KUKA KRL program: Rack_Azul_Cerrar_PLC.src, Rack_Azul_Cerrar_PLC.dat

--- Rack_Azul_Cerrar_PLC.src ---
&ACCESS RVO1
&REL 14
&COMMENT CERRAR BANDEJAS PLC
&PARAM EDITMASK = *
&PARAM TEMPLATE = C:\KRC\Roboter\Template\vorgabe
&PARAM DISKPATH = KRC:\R1\Program\MAFELEC
DEF Rack_Azul_Cerrar_PLC( )
;FOLD INI;%{PE}
  ;FOLD BASISTECH INI
    GLOBAL INTERRUPT DECL 3 WHEN $STOPMESS==TRUE DO IR_STOPM ( )
    INTERRUPT ON 3
    BAS (#INITMOV,0 )
  ;ENDFOLD (BASISTECH INI)
;FOLD SPOTTECH INI
USERSPOT(#INIT)
;ENDFOLD (SPOTTECH INI)
;FOLD GRIPPERTECH INI
USER_GRP(0,DUMMY,DUMMY,GDEFAULT)
;ENDFOLD (GRIPPERTECH INI)
  ;FOLD USER INI
    ;Make your modifications here
INTERRUPT DECL 82 WHEN I_121R1S501 DO STOP_PUSH ()
INTERRUPT DECL 92 WHEN I_121R1S501 DO STOP_PUSH ()

  ;ENDFOLD (USER INI)
;ENDFOLD (INI)
;################################################
; PROYECTO: MAFELEC PLANTA DE BATERIAS
; ROBOT: 121_R1
; PROGRAMA: CERRAR BANDEJAS EN RACK AZUL
; CREADO POR: Alejandro Company(zaisor robotics)
; FECHA: 23-NOVIEMBRE-2022
; MODIFICADO POR:
; FECHA MODIFICACION: 05-ENERO-2023
;################################################

;FOLD PTP HOME Vel=100 % PDAT1;%{PE}%R 8.3.48,%MKUKATPBASIS,%CMOVE,%VPTP,%P 1:PTP, 2:HOME, 3:, 5:100, 7:PDAT1
$BWDSTART=FALSE
PDAT_ACT=PPDAT1
FDAT_ACT=FHOME
BAS(#PTP_PARAMS,100)
$H_POS=XHOME
PTP XHOME
;ENDFOLD
; POSICION DE ESPERA ENTRADA RACK 2 (AZUL)
;FOLD PTP POS_ESPERA_AREA2 Vel=50 % H Tool[9]:T_Gripper1_Vacio Base[0];%{PE}%R 8.3.48,%MKUKATPBASIS,%CMOVE,%VPTP,%P 1:PTP, 2:POS_ESPERA_AREA2, 3:, 5:50, 7:H
$BWDSTART=FALSE
PDAT_ACT=PH
FDAT_ACT=FPOS_ESPERA_AREA2
BAS(#PTP_PARAMS,50)
PTP XPOS_ESPERA_AREA2
;ENDFOLD
;ESPERA AREA 2
WAIT FOR I_ARDY_2
O_AREL_2=FALSE

WAIT FOR I_121R1S1000==FALSE

;FOLD PTP P_CERRAR10 CONT Vel=50 % H Tool[2]:T_PUSH2 Base[2]:Rack_Azul;%{PE}%R 8.3.48,%MKUKATPBASIS,%CMOVE,%VPTP,%P 1:PTP, 2:P_CERRAR10, 3:C_DIS, 5:50, 7:H
$BWDSTART=FALSE
PDAT_ACT=PH
FDAT_ACT=FP_CERRAR10
BAS(#PTP_PARAMS,50)
PTP XP_CERRAR10 C_DIS
;ENDFOLD

INI_BUCLE:
;FOLD PTP P10 Vel=50 % H Tool[2]:T_PUSH2 Base[2]:Rack_Azul;%{PE}%R 8.3.48,%MKUKATPBASIS,%CMOVE,%VPTP,%P 1:PTP, 2:P10, 3:, 5:50, 7:H
$BWDSTART=FALSE
PDAT_ACT=PH
FDAT_ACT=FP10
BAS(#PTP_PARAMS,50)
PTP XP10
;ENDFOLD

RA_Bandeja_Nr=0
O_TYPE_RQ=TRUE
WAIT FOR (I_TYPE_INFO > 20) AND (I_TYPE_INFO < 26)
RA_Bandeja_Nr=I_TYPE_INFO

Rack_Azul_Cerrar_D ()

END
DEF STOP_PUSH()
INTERRUPT OFF 82
INTERRUPT OFF 92

BRAKE
WAIT SEC 0
PTP $POS_ACT
LIN $POS_INT
$OV_PRO=OLD_OVPRO

;RESUME

END

--- Rack_Azul_Cerrar_PLC.dat ---
&ACCESS RVO1
&REL 14
&COMMENT CERRAR BANDEJAS PLC
&PARAM EDITMASK = *
&PARAM TEMPLATE = C:\KRC\Roboter\Template\vorgabe
&PARAM DISKPATH = KRC:\R1\Program\MAFELEC
DEFDAT  Rack_Azul_Cerrar_PLC
;FOLD EXTERNAL DECLARATIONS;%{PE}%MKUKATPBASIS,%CEXT,%VCOMMON,%P
;FOLD GRIPPERTECH EXT
EXT  H50 (INT  :IN,INT  :IN,INT  :IN,GRP_TYP  :IN )
;ENDFOLD (GRIPPERTECH EXT)
;FOLD SPOTTECH EXT
EXT  USERSPOT (S_COMMAND  :IN,SPOT_TYPE  :IN )
;ENDFOLD (SPOTTECH EXT)
;FOLD BASISTECH EXT;%{PE}%MKUKATPBASIS,%CEXT,%VEXT,%P
EXT  BAS (BAS_COMMAND  :IN,REAL  :IN )
DECL INT SUCCESS
;ENDFOLD (BASISTECH EXT)
;FOLD USER EXT;%{E}%MKUKATPUSER,%CEXT,%VEXT,%P
;Make your modifications here

;ENDFOLD (USER EXT)
;ENDFOLD (EXTERNAL DECLARATIONS)
DECL BASIS_SUGG_T LAST_BASIS={POINT1[] "HOME                    ",POINT2[] "HOME                    ",CP_PARAMS[] "CPDAT0                  ",PTP_PARAMS[] "PDAT1                   ",CONT[] "                        ",CP_VEL[] "2.0                     ",PTP_VEL[] "100                     ",SYNC_PARAMS[] "SYNCDAT                 ",SPL_NAME[] "S0                      ",A_PARAMS[] "ADAT0                   "}
DECL PDAT PH={VEL 100.000,ACC 100.000,APO_DIST 100.000,APO_MODE #CDIS,GEAR_JERK 50.0000,EXAX_IGN 0}
DECL E6POS XPOS_ESPERA_AREA1={X 112.943756,Y -227.851166,Z 2716.11304,A 36.2463837,B -15.5853510,C 56.0520973,S 3,T 42,E1 0.0,E2 0.0,E3 0.0,E4 0.0,E5 0.0,E6 0.0}
DECL FDAT FPOS_ESPERA_AREA1={TOOL_NO 9,BASE_NO 0,IPO_FRAME #BASE,POINT2[] " ",TQ_STATE FALSE}
DECL LDAT LL={VEL 2.00000,ACC 25.0000,APO_DIST 25.0000,APO_FAC 50.0000,AXIS_VEL 100.000,AXIS_ACC 100.000,ORI_TYP #VAR,CIRC_TYP #BASE,JERK_FAC 50.0000,GEAR_JERK 50.0000,EXAX_IGN 0}
DECL E6POS XPOS_AREA1_LIBRE={X -250.533554,Y -43.6507149,Z 2716.11304,A -84.6604385,B 6.50295877,C 57.2217522,S 3,T 42,E1 0.0,E2 0.0,E3 0.0,E4 0.0,E5 0.0,E6 0.0}
DECL FDAT FPOS_AREA1_LIBRE={TOOL_NO 9,BASE_NO 0,IPO_FRAME #BASE,POINT2[] " ",TQ_STATE FALSE}
DECL E6POS XP111={X 557.799622,Y -753.947571,Z -222.785736,A -88.9974060,B 13.7721291,C 89.1738281,S 6,T 58,E1 0.0,E2 0.0,E3 0.0,E4 0.0,E5 0.0,E6 0.0}
DECL FDAT FP111={TOOL_NO 1,BASE_NO 1,IPO_FRAME #BASE,POINT2[] " ",TQ_STATE FALSE}
DECL E6POS XP10={X 1430.18262,Y 33.1879578,Z 909.224609,A 86.6829224,B -17.0911541,C -157.124573,S 2,T 35,E1 0.0,E2 0.0,E3 0.0,E4 0.0,E5 0.0,E6 0.0}
DECL FDAT FP10={TOOL_NO 2,BASE_NO 2,IPO_FRAME #BASE,POINT2[] " ",TQ_STATE FALSE}
DECL E6POS XP110={X 632.645691,Y 303.475861,Z -186.174820,A -88.8950272,B 31.1322117,C 89.5053635,S 6,T 58,E1 0.0,E2 0.0,E3 0.0,E4 0.0,E5 0.0,E6 0.0}
DECL FDAT FP110={TOOL_NO 1,BASE_NO 1,IPO_FRAME #BASE,POINT2[] " ",TQ_STATE FALSE}
DECL E6POS XP120={X 535.775818,Y 225.276917,Z -536.621948,A -91.0083771,B 14.9493265,C 94.2730637,S 6,T 58,E1 0.0,E2 0.0,E3 0.0,E4 0.0,E5 0.0,E6 0.0}
DECL FDAT FP120={TOOL_NO 1,BASE_NO 1,IPO_FRAME #BASE,POINT2[] " ",TQ_STATE FALSE}
DECL E6POS XP_ABRIR10={X -250.533554,Y -43.6507149,Z 2716.11304,A -84.6604385,B 6.50295877,C 57.2217522,S 3,T 42,E1 0.0,E2 0.0,E3 0.0,E4 0.0,E5 0.0,E6 0.0}
DECL FDAT FP_ABRIR10={TOOL_NO 9,BASE_NO 0,IPO_FRAME #BASE,POINT2[] " ",TQ_STATE FALSE}
DECL E6POS XP_AHOME={X 112.943756,Y -227.851166,Z 2716.11304,A 36.2463837,B -15.5853510,C 56.0520973,S 3,T 42,E1 0.0,E2 0.0,E3 0.0,E4 0.0,E5 0.0,E6 0.0}
DECL FDAT FP_aHOME={TOOL_NO 9,BASE_NO 0,IPO_FRAME #BASE,POINT2[] " ",TQ_STATE FALSE}
DECL E6POS XIni_Cerrar_B1={X 557.764587,Y -781.945251,Z -181.205933,A -89.0119858,B 10.6981707,C 89.1186752,S 6,T 58,E1 0.0,E2 0.0,E3 0.0,E4 0.0,E5 0.0,E6 0.0}
DECL FDAT FIni_Cerrar_B1={TOOL_NO 1,BASE_NO 1,IPO_FRAME #BASE,POINT2[] " ",TQ_STATE FALSE}
DECL E6POS XAux_Cerrar_B1={X 557.840454,Y -622.833801,Z -384.869720,A -88.9527512,B 18.9294662,C 89.2742310,S 6,T 58,E1 0.0,E2 0.0,E3 0.0,E4 0.0,E5 0.0,E6 0.0}
DECL E6POS XFin_Cerrar_B1={X 558.459229,Y -381.955719,Z -941.239441,A -88.7644653,B 34.8009872,C 89.6337738,S 6,T 58,E1 0.0,E2 0.0,E3 0.0,E4 0.0,E5 0.0,E6 0.0}
DECL FDAT FFin_Cerrar_B1={TOOL_NO 1,BASE_NO 1,IPO_FRAME #BASE,POINT2[] "XAux_Cerrar_B1",TQ_STATE FALSE}
DECL E6POS XP0={X 632.645691,Y 303.475861,Z -186.174820,A -88.8950272,B 31.1322117,C 89.5053635,S 6,T 58,E1 0.0,E2 0.0,E3 0.0,E4 0.0,E5 0.0,E6 0.0}
DECL FDAT FP0={TOOL_NO 1,BASE_NO 1,IPO_FRAME #BASE,POINT2[] " ",TQ_STATE FALSE}
DECL E6POS XIni_Cerrar_B2={X 633.606323,Y -740.251,Z 3.60236120,A -89.0051498,B 9.17837143,C 89.0890656,S 6,T 58,E1 0.0,E2 0.0,E3 0.0,E4 0.0,E5 0.0,E6 0.0}
DECL FDAT FIni_Cerrar_B2={TOOL_NO 1,BASE_NO 1,IPO_FRAME #BASE,POINT2[] " ",TQ_STATE FALSE}
DECL E6POS XP1={X 633.606323,Y -740.251,Z -11.7250,A -89.0051498,B 9.17837143,C 89.0890656,S 6,T 58,E1 0.0,E2 0.0,E3 0.0,E4 0.0,E5 0.0,E6 0.0}
DECL FDAT FP1={TOOL_NO 1,BASE_NO 1,IPO_FRAME #BASE,POINT2[] " ",TQ_STATE FALSE}
DECL E6POS XAux_Cerrar_B2={X 634.042603,Y -508.122833,Z -357.182983,A -88.8871536,B 26.3570118,C 89.4227295,S 6,T 58,E1 0.0,E2 0.0,E3 0.0,E4 0.0,E5 0.0,E6 0.0}
DECL E6POS XFin_Cerrar_B2={X 634.405884,Y -397.733490,Z -741.710266,A -88.8505630,B 28.6699753,C 89.4738922,S 6,T 58,E1 0.0,E2 0.0,E3 0.0,E4 0.0,E5 0.0,E6 0.0}
DECL FDAT FFin_Cerrar_B2={TOOL_NO 1,BASE_NO 1,IPO_FRAME #BASE,POINT2[] "XAux_Cerrar_B2",TQ_STATE FALSE}
DECL E6POS XP2={X 535.775818,Y 225.276917,Z -536.621948,A -91.0083771,B 14.9493265,C 94.2730637,S 6,T 58,E1 0.0,E2 0.0,E3 0.0,E4 0.0,E5 0.0,E6 0.0}
DECL FDAT FP2={TOOL_NO 1,BASE_NO 1,IPO_FRAME #BASE,POINT2[] " ",TQ_STATE FALSE}
DECL E6POS XP210={X 536.241516,Y 225.176605,Z 24.6719704,A -90.9851761,B 14.9447651,C 94.2668762,S 6,T 58,E1 0.0,E2 0.0,E3 0.0,E4 0.0,E5 0.0,E6 0.0}
DECL FDAT FP210={TOOL_NO 1,BASE_NO 1,IPO_FRAME #BASE,POINT2[] " ",TQ_STATE FALSE}
DECL E6POS XP220={X 535.775818,Y 225.276917,Z -194.099075,A -91.0083771,B 14.9493265,C 94.2730637,S 6,T 58,E1 0.0,E2 0.0,E3 0.0,E4 0.0,E5 0.0,E6 0.0}
DECL FDAT FP220={TOOL_NO 1,BASE_NO 1,IPO_FRAME #BASE,POINT2[] " ",TQ_STATE FALSE}
DECL E6POS XP3={X 536.241516,Y 225.176605,Z 24.6719704,A -90.9851761,B 14.9447651,C 94.2668762,S 6,T 58,E1 0.0,E2 0.0,E3 0.0,E4 0.0,E5 0.0,E6 0.0}
DECL FDAT FP3={TOOL_NO 1,BASE_NO 1,IPO_FRAME #BASE,POINT2[] " ",TQ_STATE FALSE}
DECL E6POS XIni_Cerrar_B3={X 587.397888,Y -796.521118,Z 250.544754,A -89.9228,B 6.59320593,C 91.5957413,S 6,T 58,E1 0.0,E2 0.0,E3 0.0,E4 0.0,E5 0.0,E6 0.0}
DECL FDAT FIni_Cerrar_B3={TOOL_NO 1,BASE_NO 1,IPO_FRAME #BASE,POINT2[] " ",TQ_STATE FALSE}
DECL E6POS XP4={X 633.606323,Y -740.251,Z -11.7250,A -89.0051498,B 9.17837143,C 89.0890656,S 6,T 58,E1 0.0,E2 0.0,E3 0.0,E4 0.0,E5 0.0,E6 0.0}
DECL FDAT FP4={TOOL_NO 1,BASE_NO 1,IPO_FRAME #BASE,POINT2[] " ",TQ_STATE FALSE}
DECL E6POS XAux_Cerrar_B3={X 587.803650,Y -538.859497,Z -87.8424835,A -89.9063950,B 15.5115423,C 91.6123123,S 6,T 58,E1 0.0,E2 0.0,E3 0.0,E4 0.0,E5 0.0,E6 0.0}
DECL E6POS XFin_Cerrar_B3={X 588.007202,Y -397.554932,Z -533.267273,A -89.8953171,B 21.9562569,C 91.6268768,S 6,T 58,E1 0.0,E2 0.0,E3 0.0,E4 0.0,E5 0.0,E6 0.0}
DECL FDAT FFin_Cerrar_B3={TOOL_NO 1,BASE_NO 1,IPO_FRAME #BASE,POINT2[] "XAux_Cerrar_B3",TQ_STATE FALSE}
DECL E6POS XP5={X 535.775818,Y 225.276917,Z -194.099075,A -91.0083771,B 14.9493265,C 94.2730637,S 6,T 58,E1 0.0,E2 0.0,E3 0.0,E4 0.0,E5 0.0,E6 0.0}
DECL FDAT FP5={TOOL_NO 1,BASE_NO 1,IPO_FRAME #BASE,POINT2[] " ",TQ_STATE FALSE}
DECL E6POS XP310={X 536.344910,Y 225.151108,Z 251.906281,A -90.9788437,B 14.9441595,C 94.2655792,S 6,T 26,E1 0.0,E2 0.0,E3 0.0,E4 0.0,E5 0.0,E6 0.0}
DECL FDAT FP310={TOOL_NO 1,BASE_NO 1,IPO_FRAME #BASE,POINT2[] " ",TQ_STATE FALSE}
DECL E6POS XP320={X 535.775818,Y 225.276917,Z -194.099075,A -91.0083771,B 14.9493265,C 94.2730637,S 6,T 58,E1 0.0,E2 0.0,E3 0.0,E4 0.0,E5 0.0,E6 0.0}
DECL FDAT FP320={TOOL_NO 1,BASE_NO 1,IPO_FRAME #BASE,POINT2[] " ",TQ_STATE FALSE}
DECL E6POS XP310_1={X 587.398743,Y -796.520813,Z 219.048569,A -89.9227676,B 6.59320068,C 91.5957413,S 6,T 58,E1 0.0,E2 0.0,E3 0.0,E4 0.0,E5 0.0,E6 0.0}
DECL FDAT FP310_1={TOOL_NO 1,BASE_NO 1,IPO_FRAME #BASE,POINT2[] " ",TQ_STATE FALSE}
DECL E6POS XP6={X 536.241516,Y 225.176605,Z 24.6719704,A -90.9851761,B 14.9447651,C 94.2668762,S 6,T 58,E1 0.0,E2 0.0,E3 0.0,E4 0.0,E5 0.0,E6 0.0}
DECL FDAT FP6={TOOL_NO 1,BASE_NO 1,IPO_FRAME #BASE,POINT2[] " ",TQ_STATE FALSE}
DECL E6POS XIni_Cerrar_B4={X 547.014465,Y -762.279480,Z 527.953308,A -92.0144501,B 13.7285652,C 90.3226547,S 6,T 26,E1 0.0,E2 0.0,E3 0.0,E4 0.0,E5 0.0,E6 0.0}
DECL FDAT FIni_Cerrar_B4={TOOL_NO 1,BASE_NO 1,IPO_FRAME #BASE,POINT2[] " ",TQ_STATE FALSE}
DECL E6POS XP7={X 633.606323,Y -740.251,Z -11.7250,A -89.0051498,B 9.17837143,C 89.0890656,S 6,T 58,E1 0.0,E2 0.0,E3 0.0,E4 0.0,E5 0.0,E6 0.0}
DECL FDAT FP7={TOOL_NO 1,BASE_NO 1,IPO_FRAME #BASE,POINT2[] " ",TQ_STATE FALSE}
DECL E6POS XAux_Cerrar_B4={X 547.619568,Y -529.437683,Z 86.4444046,A -92.0362,B 21.7243443,C 90.2498322,S 6,T 26,E1 0.0,E2 0.0,E3 0.0,E4 0.0,E5 0.0,E6 0.0}
DECL E6POS XFin_Cerrar_B4={X 547.891113,Y -426.606598,Z -334.407837,A -92.0266571,B 21.7223244,C 90.2480469,S 6,T 58,E1 0.0,E2 0.0,E3 0.0,E4 0.0,E5 0.0,E6 0.0}
DECL FDAT FFin_Cerrar_B4={TOOL_NO 1,BASE_NO 1,IPO_FRAME #BASE,POINT2[] "XAux_Cerrar_B4",TQ_STATE FALSE}
DECL E6POS XP8={X 535.775818,Y 225.276917,Z -194.099075,A -91.0083771,B 14.9493265,C 94.2730637,S 6,T 58,E1 0.0,E2 0.0,E3 0.0,E4 0.0,E5 0.0,E6 0.0}
DECL FDAT FP8={TOOL_NO 1,BASE_NO 1,IPO_FRAME #BASE,POINT2[] " ",TQ_STATE FALSE}
DECL E6POS XP410={X 546.439087,Y 225.985733,Z 608.963928,A -94.2845764,B 13.2172089,C 80.7249,S 6,T 26,E1 0.0,E2 0.0,E3 0.0,E4 0.0,E5 0.0,E6 0.0}
DECL FDAT FP410={TOOL_NO 1,BASE_NO 1,IPO_FRAME #BASE,POINT2[] " ",TQ_STATE FALSE}
DECL E6POS XP410_1={X 547.319458,Y -761.898315,Z 410.812561,A -92.0465546,B 21.7247772,C 90.2501144,S 6,T 26,E1 0.0,E2 0.0,E3 0.0,E4 0.0,E5 0.0,E6 0.0}
DECL FDAT FP410_1={TOOL_NO 1,BASE_NO 1,IPO_FRAME #BASE,POINT2[] " ",TQ_STATE FALSE}
DECL E6POS XP420={X 525.192,Y 187.708069,Z 115.738434,A -91.6678391,B 6.13838816,C 94.1520309,S 6,T 58,E1 0.0,E2 0.0,E3 0.0,E4 0.0,E5 0.0,E6 0.0}
DECL FDAT FP420={TOOL_NO 1,BASE_NO 1,IPO_FRAME #BASE,POINT2[] " ",TQ_STATE FALSE}
DECL E6POS XP9={X 536.241516,Y 225.176605,Z 24.6719704,A -90.9851761,B 14.9447651,C 94.2668762,S 6,T 58,E1 0.0,E2 0.0,E3 0.0,E4 0.0,E5 0.0,E6 0.0}
DECL FDAT FP9={TOOL_NO 1,BASE_NO 1,IPO_FRAME #BASE,POINT2[] " ",TQ_STATE FALSE}
DECL E6POS XIni_Cerrar_B5={X 644.333130,Y -771.042114,Z 1009.38544,A -93.7095184,B 18.5084820,C 84.4919510,S 6,T 26,E1 0.0,E2 0.0,E3 0.0,E4 0.0,E5 0.0,E6 0.0}
DECL FDAT FIni_Cerrar_B5={TOOL_NO 1,BASE_NO 1,IPO_FRAME #BASE,POINT2[] " ",TQ_STATE FALSE}
DECL E6POS XP11={X 633.606323,Y -740.251,Z -11.7250,A -89.0051498,B 9.17837143,C 89.0890656,S 6,T 58,E1 0.0,E2 0.0,E3 0.0,E4 0.0,E5 0.0,E6 0.0}
DECL FDAT FP11={TOOL_NO 1,BASE_NO 1,IPO_FRAME #BASE,POINT2[] " ",TQ_STATE FALSE}
DECL E6POS XAux_Cerrar_B5={X 645.412,Y -297.960297,Z 334.856628,A -91.5430527,B 23.7528038,C 84.3394470,S 6,T 26,E1 0.0,E2 0.0,E3 0.0,E4 0.0,E5 0.0,E6 0.0}
DECL E6POS XFin_Cerrar_B5={X 647.239136,Y -199.588867,Z -115.631508,A -87.2260361,B 11.0592718,C 90.0945892,S 6,T 58,E1 0.0,E2 0.0,E3 0.0,E4 0.0,E5 0.0,E6 0.0}
DECL FDAT FFin_Cerrar_B5={TOOL_NO 1,BASE_NO 1,IPO_FRAME #BASE,POINT2[] "XAux_Cerrar_B5",TQ_STATE FALSE}
DECL E6POS XP12={X 535.775818,Y 225.276917,Z -194.099075,A -91.0083771,B 14.9493265,C 94.2730637,S 6,T 58,E1 0.0,E2 0.0,E3 0.0,E4 0.0,E5 0.0,E6 0.0}
DECL FDAT FP12={TOOL_NO 1,BASE_NO 1,IPO_FRAME #BASE,POINT2[] " ",TQ_STATE FALSE}
DECL E6POS XP510={X 642.977051,Y 234.134598,Z 1082.35,A -97.9549866,B 9.71833515,C 62.4231300,S 6,T 26,E1 0.0,E2 0.0,E3 0.0,E4 0.0,E5 0.0,E6 0.0}
DECL FDAT FP510={TOOL_NO 1,BASE_NO 1,IPO_FRAME #BASE,POINT2[] " ",TQ_STATE FALSE}
DECL E6POS XP510_1={X 644.512329,Y -684.707275,Z 831.107483,A -91.5230255,B 18.5093899,C 84.4910736,S 6,T 26,E1 0.0,E2 0.0,E3 0.0,E4 0.0,E5 0.0,E6 0.0}
DECL FDAT FP510_1={TOOL_NO 1,BASE_NO 1,IPO_FRAME #BASE,POINT2[] " ",TQ_STATE FALSE}
DECL E6POS XP520={X 536.730957,Y 225.074142,Z 89.3547668,A -90.9613,B 14.9400396,C 94.2604446,S 6,T 58,E1 0.0,E2 0.0,E3 0.0,E4 0.0,E5 0.0,E6 0.0}
DECL FDAT FP520={TOOL_NO 1,BASE_NO 1,IPO_FRAME #BASE,POINT2[] " ",TQ_STATE FALSE}
DECL E6POS XP210_1={X 633.606323,Y -740.251,Z -11.7250,A -89.0051498,B 9.17837143,C 89.0890656,S 6,T 58,E1 0.0,E2 0.0,E3 0.0,E4 0.0,E5 0.0,E6 0.0}
DECL FDAT FP210_1={TOOL_NO 1,BASE_NO 1,IPO_FRAME #BASE,POINT2[] " ",TQ_STATE FALSE}
DECL E6POS XP110_1={X 557.799622,Y -753.947571,Z -222.785736,A -88.9974060,B 13.7721291,C 89.1738281,S 6,T 58,E1 0.0,E2 0.0,E3 0.0,E4 0.0,E5 0.0,E6 0.0}
DECL FDAT FP110_1={TOOL_NO 1,BASE_NO 1,IPO_FRAME #BASE,POINT2[] " ",TQ_STATE FALSE}
DECL E6POS XP_FIN={X 536.730957,Y 225.074142,Z 89.3547668,A -90.9613,B 14.9400396,C 94.2604446,S 6,T 58,E1 0.0,E2 0.0,E3 0.0,E4 0.0,E5 0.0,E6 0.0}
DECL FDAT FP_FIN={TOOL_NO 2,BASE_NO 2,IPO_FRAME #BASE,POINT2[] " ",TQ_STATE FALSE}
DECL E6POS XP_CERRAR10={X 2082.73657,Y -449.358490,Z 1844.21362,A 56.4428596,B -36.9036674,C -95.8930435,S 2,T 35,E1 0.0,E2 0.0,E3 0.0,E4 0.0,E5 0.0,E6 0.0}
DECL FDAT FP_CERRAR10={TOOL_NO 2,BASE_NO 2,IPO_FRAME #BASE,POINT2[] " ",TQ_STATE FALSE}
DECL E6POS XPOS_AREA2_LIBRE={X -250.533554,Y -43.6507149,Z 2716.11304,A -84.6604385,B 6.50295877,C 57.2217522,S 3,T 42,E1 0.0,E2 0.0,E3 0.0,E4 0.0,E5 0.0,E6 0.0}
DECL FDAT FPOS_AREA2_LIBRE={TOOL_NO 9,BASE_NO 0,IPO_FRAME #BASE,POINT2[] " ",TQ_STATE FALSE}
DECL E6POS XPOS_ESPERA_AREA2={X 336.434082,Y 138.108124,Z 2801.35059,A 102.311447,B 52.9667473,C 77.5465240,S 2,T 35,E1 0.0,E2 0.0,E3 0.0,E4 0.0,E5 0.0,E6 0.0}
DECL FDAT FPOS_ESPERA_AREA2={TOOL_NO 9,BASE_NO 0,IPO_FRAME #BASE,POINT2[] " ",TQ_STATE FALSE}
DECL PDAT PPDAT1={VEL 100.000,ACC 100.000,APO_DIST 100.000,GEAR_JERK 50.0000,EXAX_IGN 0}
ENDDAT
